// TwinCAT 3 PLC project SPS1
// ProgramVersion: 3.1.4023.0
// libraries:
//   Tc2_MC2, * (Beckhoff Automation GmbH)
//   Tc2_MC2_Drive, * (Beckhoff Automation GmbH)
//   Tc2_Standard, * (Beckhoff Automation GmbH)
//   Tc2_System, * (Beckhoff Automation GmbH)
//   Tc2_Utilities, * (Beckhoff Automation GmbH)
//   Tc3_Module, * (Beckhoff Automation GmbH)
//   Tc3_System, * (Beckhoff Automation GmbH)
// project tree:
//   DUTs/Standard/FunE/ u_FunEIF.TcDUT, u_FunEIF_In.TcDUT, u_FunEIF_InOut.TcDUT, u_FunEIF_Out.TcDUT, u_FunEIF_Stat.TcDUT
//   GVLs/Standard/ DB_FunE_IF.TcGVL, Globale_Konstanten.TcGVL
//   / PlcTask.TcTTO
//   POUs/ MAIN.TcPOU
//   POUs/Standardt/Hilfsfunktionen Zeit/ R_SYS_T.TcPOU, T_DIFF.TcPOU
//   POUs/Standardt/Zentral/ FB_Zentral.TcPOU, FB_Zentral_TaktimpulsGenerator.TcPOU
// real-time tasks:
//   TASK PlcTask: cycle T#10ms, priority 20, ADS port 350
// I/O:
//   DEVICE Gerät 1 (EtherCAT) (disabled), AmsNetId 192.168.27.57.2.1
//     Klemme 1 (EK1100) [EK1100 EtherCAT-Koppler (2A E-Bus)]
//       Klemme 2 (EL7201) [EL7201 1K. MDP742 Servo-Motor-Endstufe (50V, 4A)]

CONFIGURATION SPS1
    RESOURCE PLC ON TwinCAT3
        TASK PlcTask(INTERVAL := T#10ms, PRIORITY := 20);
        PROGRAM MAIN WITH PlcTask : MAIN;
    END_RESOURCE
END_CONFIGURATION

// ---- DUTs/Standard/FunE/u_FunEIF.TcDUT
TYPE u_FunEIF :
STRUCT
	I									:u_FunEIF_In; 
	O									:u_FunEIF_Out; 
	X									:u_FunEIF_InOut;
	Stat								:u_FunEIF_Stat;
END_STRUCT
END_TYPE

// ---- DUTs/Standard/FunE/u_FunEIF_In.TcDUT
TYPE u_FunEIF_In :
STRUCT
	x_Start									:BOOL := FALSE;															//Start Ablauf
	x_Init									:BOOL := FALSE; 														//Anwahl Initialisierung
	x_Freigabe							:BOOL := FALSE; 														//Freigabe Ablauf
	x_FreigabeHalt						:BOOL := FALSE; 														//Freigabe Unterbrechung
	x_FreigabeStoerung			:BOOL := FALSE; 														//Freigabe Stoerung
	x_FreigabeZeitEinlernen		:BOOL := FALSE; 														//Freigabe Ermittlung Regelzeit
	x_uFunEGST							:BOOL := FALSE; 														//unterlagerte Funktionselemente : alle in Grundstellungs
	x_uFunEinitAktiv					:BOOL := FALSE; 														//unterlagerte Funktionselemente: mind. 1 initialisierung aktiv 
	x_uFunEHalt							:BOOL := FALSE; 														//unterlagerte Funktionselemente: mind. 1 noch nicht fertig
	x_uFunEStoerung				:BOOL := FALSE; 														//unterlagerte Funktionselemente: mind. 1 hat Stoerung
	x_SimulationAktiv					:BOOL := FALSE; 														//Simulation aktiv
	i_Auftrag								:BOOL := FALSE; 														//Auftragsnummer
	t_Simulationszeit					:TIME := T#1S; 															//Verzögerungszeit für Simulation
	t_TimeOut							:TIME := T#1S; 															//TimeOut für Meldung wenn FunE länger braucht als eingelernt
	s_Name								:STRING := "Kein Funktionselement vergeben"; 		//Name des Funktionselements
	i_FunETyp							:INT := 0; 																	//Typ/Art des Funktionselements
	i_MasterFunE						:INT := 0; 																	//uebergeordnetes Funktionselement (bei 0 kein uebergeordnetes FunE)
END_STRUCT
END_TYPE

// ---- DUTs/Standard/FunE/u_FunEIF_InOut.TcDUT
TYPE u_FunEIF_InOut :
STRUCT
	x_Parameter					:ARRAY[0..255] OF BOOL; 
	di_Parameter					:ARRAY[0..31] OF DINT; 
	lr_Parameter					:ARRAY[0..31] OF LREAL; 
	s_Parameter					:ARRAY[0..1] OF STRING; 
END_STRUCT
END_TYPE

// ---- DUTs/Standard/FunE/u_FunEIF_Out.TcDUT
TYPE u_FunEIF_Out :
STRUCT
	x_bereit								:BOOL :=FALSE; 													//Funktionselement ist bereit
	x_arbeitet							:BOOL :=FALSE; 													//Funktionselement arbeitet
	x_fertig								:BOOL :=FALSE; 													//Funktionselement hat Zyklus beendet (steht bis zum nächsten Zyklus an)
	x_Fehler								:BOOL :=FALSE; 													//Funktionselement hat Fehler
	x_Grundstellung					:BOOL :=FALSE; 													//Funktionselement ist in Grundstellung
	x_initAktiv							:BOOL :=FALSE; 													//Funktionselement initialisierung aktiv 
	s_Aktionsname					:STRING :=""; 													//Name der aktuellen Aktion
	di_Status								:DINT := 0; 															//Statuscode (negativ=Fehler/positiv=erfolgreich)
	t_ZeitLetzerZyklus				:TIME := T#0MS; 												//Bearbeitungszeit letzter Ablauf
	di_Aktivierungen					:DINT := 0; 															//Anzahl der Aktivierungen 
	lt_Betriebsstundenzaehler 	:LTIME := LTIME#0MS; 										//Betriebsstundenzaehler
END_STRUCT
END_TYPE

// ---- DUTs/Standard/FunE/u_FunEIF_Stat.TcDUT
TYPE u_FunEIF_Stat :
STRUCT
	x_Halt												:BOOL :=FALSE; 								//FunE Halt
	x_Betrieb											:BOOL :=FALSE; 								//Betriebsfreigabe
	x_WSB												:BOOL :=FALSE;								//Weiterschaltbedingung
	x_Schrittwechsel								:BOOL :=FALSE; 								//Schrittwechsel aktiv
	i_SchrittFlanke									:INT :=0; 										//Schritt letzter SPS - Zyklus (benötigt zur Erkennung des Schrittwechsels)
	i_Schritt											:INT:= 0; 										//aktueller Schritt der Schrittkette
	i_SchrittAlt										:INT :=0; 										//letzter Schritt
	dt_StartZeit										:DT := DT#1972-03-29-00:00:00;	//Zeit, an dem das Funktionselement gestartet wurde	(Achtung!!!: In DT sind im gegensatz zu Siemens keine MS enthalten!!!)
	dt_LaufzeitFunE								:DT := DT#1972-03-29-00:00:00;  	//Zeit seit Start des Funktionselements (Achtung!!!: In DT sind im gegensatz zu Siemens keine MS enthalten!!!)
	t_mittlereZykluszeit							:TIME :=T#0MS; 								//eingelernte Zykluszeit
	o_Simulationszeit								:TON; 												//Timer für die Simulation des Funktionselements
END_STRUCT
END_TYPE

// ---- GVLs/Standard/DB_FunE_IF.TcGVL
{attribute 'qualified_only'}
VAR_GLOBAL
	Nr																	:ARRAY[0..Globale_Konstanten.Ci_Funktionselmente] OF u_FunEIF; 
	Anwahl_HMI_FunE_1									:INT :=0; 
	Anwahl_HMI_FunE_2									:INT :=0; 
	Anwahl_HMI_FunE_3									:INT :=0; 
	Anwahl_HMI_FunE_4									:INT :=0; 
END_VAR

// ---- GVLs/Standard/Globale_Konstanten.TcGVL
{attribute 'qualified_only'}
//Anwenderkonstanten
VAR_GLOBAL CONSTANT
	Ci_ZentralModuleAnzahl				:INT 		:=1; 					//Anzahl der autarken Zentralmodule
	Ci_Funktionselmente					:INT 		:=999; 				//Anzahl der Funktionselemente 
	Ci_Mod1										:INT			:=1; 					//EnumMR - Modul1
	Ci_Mod1RT1									:INT			:=1; 					//EnumMR - Modul1 RT1
END_VAR

// ---- POUs/MAIN.TcPOU
PROGRAM MAIN
VAR
	So_Taktgenerator				: FB_Zentral_TaktimpulsGenerator; 
	
	Sx_Takt			: BOOL; 
	Sx_Impuls		: BOOL; 
	Si_Counter		: INT; 
	
END_VAR


So_Taktgenerator(Ir_Frequenz := 1.0, Ox_Takt => Sx_Takt, Ox_Impuls => Sx_Impuls); 

IF(Sx_Impuls) THEN 
	Si_Counter := Si_Counter + 1;
END_IF

END_PROGRAM

// ---- POUs/Standardt/Zentral/FB_Zentral_TaktimpulsGenerator.TcPOU
FUNCTION_BLOCK FB_Zentral_TaktimpulsGenerator
VAR_INPUT
	Ir_Frequenz		: REAL; 
END_VAR
VAR_OUTPUT
	Ox_Takt								: BOOL; 
	Ox_Impuls							: BOOL; 
END_VAR

VAR
	St_TakttimerEinfach					: TON; 
	ReadRTC									: R_SYS_T; 
	TimeValid									: BOOL; 
	RTCTime									: DT; 
	RTCMillis									: DWORD; 
	Sdt_StartAktuellerTakt				: DT; 
	Sx_TaktFP								: BOOL; 
	Sx_Init										: BOOL; 
	St_DifferenzStartAktuell			:TIME; 	
	Sdw_StartAktuellerTaktMillis	:DWORD;  
END_VAR
	
VAR_TEMP

END_VAR

//Erfassung aktuelle Date and Time
ReadRTC(It_SynchTime := T#5S, Ox_TimeValid => TimeValid, Odt_RTCTime => RTCTime, Odw_Milliseconds => RTCMillis);  
	
//Ermittlung Dauer seit Taktstart
St_DifferenzStartAktuell := T_DIFF(Idt_Time1 := RTCTime, Idw_Time1Millis :=RTCMillis, Idt_Time2 := Sdt_StartAktuellerTakt, Idw_Time2Millis := Sdw_StartAktuellerTaktMillis); 


//Taktbildung (halbe Zeit an/ halbe Zeit aus)
Ox_Takt := St_DifferenzStartAktuell > DINT_TO_TIME(REAL_TO_DINT((1000/Ir_Frequenz)/2)); 
	
//Impuls Takt 
Ox_Impuls := Ox_Takt AND NOT Sx_TaktFP;
Sx_TaktFP := Ox_Takt; 
	
//Abspeichern Start aktueller Takt
IF (St_DifferenzStartAktuell > DINT_TO_TIME(REAL_TO_DINT((1000/Ir_Frequenz)))) OR NOT Sx_Init THEN 
	Sdt_StartAktuellerTakt := RTCTime; 
	Sdw_StartAktuellerTaktMillis := RTCMillis; 
END_IF
	
//Baustein als initialisiert setzen 
Sx_Init := TRUE;

END_FUNCTION_BLOCK

// ---- POUs/Standardt/Hilfsfunktionen Zeit/R_SYS_T.TcPOU
FUNCTION_BLOCK R_SYS_T
VAR_INPUT
	It_SynchTime						: TIME; 
END_VAR
VAR_OUTPUT
	Odt_RTCTime						: DT; 
	Odw_Milliseconds					: DWORD; 
	Ox_TimeValid						: BOOL; 
END_VAR
VAR
	So_SynchronizeTimer			: TON; 
	So_ReadSystemTime			: NT_GetTime; 
	Ss_SystemTime					: TIMESTRUCT; 
	Sx_Synch								: BOOL; 
	So_SynchTrigger					: F_TRIG; 
	So_RTC								: RTC_EX; 
	
	//Debug variables
	Si_SynchCounter					: DWORD; 
	
END_VAR

//Defines
{define DEBUG}

//Read System Time cyclic with period based on the Synch time 
So_SynchronizeTimer(IN := NOT So_SynchronizeTimer.Q, PT := It_SynchTime);
So_ReadSystemTime(START := So_SynchronizeTimer.Q,  TMOUT := DEFAULT_ADS_TIMEOUT, TIMESTR => Ss_SystemTime); 

//Create the synchronise bit
So_SynchTrigger(CLK := (So_ReadSystemTime.BUSY AND NOT So_ReadSystemTime.ERR)); 

//Count the Synchs in Debug Mode
{IF defined (DEBUG)}
	IF(So_SynchTrigger.Q) THEN 
		Si_SynchCounter := Si_SynchCounter + 1; 
	END_IF
{END_IF}

//RTC Synchronisieren und auslesen 
So_RTC(EN := So_SynchTrigger.Q, PDT := SYSTEMTIME_TO_DT(Ss_SystemTime), PMSEK := Ss_SystemTime.wMilliseconds, Q => Ox_TimeValid, CDT => Odt_RTCTime, CMSEK => Odw_Milliseconds);

END_FUNCTION_BLOCK

// ---- POUs/Standardt/Hilfsfunktionen Zeit/T_DIFF.TcPOU
FUNCTION T_DIFF : Time
VAR_INPUT
	Idt_Time1				:DT; 
	Idw_Time1Millis	:DWORD; 
	Idt_Time2				:DT; 
	Idw_Time2Millis	:DWORD; 
END_VAR
VAR
	Ss_Time1						:TIMESTRUCT;
	Ss_Time2						:TIMESTRUCT;
	Sw_HourDiff					:WORD; 
	Sw_MinuteDiff				:WORD; 
	Sw_SecondDiff				:WORD; 
	Sw_MillisecondsDiff		:DWORD;
	Sdw_TimeInMillis			:DWORD ; 
END_VAR

//Convert the time to TIMESTRUCT
Ss_Time1 := DT_TO_SYSTEMTIME(Idt_Time1); 
Ss_Time2 := DT_TO_SYSTEMTIME(Idt_Time2); 

//Subract
Sw_HourDiff := Ss_Time1.wHour - Ss_Time2.wHour; 
Sw_MinuteDiff := Ss_Time1.wMinute - Ss_Time2.wMinute; 
Sw_SecondDiff := Ss_Time1.wSecond - Ss_Time2.wSecond; 
Sw_MillisecondsDiff := Idw_Time1Millis - Idw_Time2Millis;

//Convert to millis
Sdw_TimeInMillis := Sdw_TimeInMillis + Sw_MillisecondsDiff; 
Sdw_TimeInMillis := Sdw_TimeInMillis + (Sw_SecondDiff*1000);
Sdw_TimeInMillis := Sdw_TimeInMillis + (Sw_MinuteDiff*1000*60); 
Sdw_TimeInMillis := Sdw_TimeInMillis + (Sw_HourDiff*1000*60*60); 

//Return 
T_DIFF := DWORD_TO_TIME(Sdw_TimeInMillis);

END_FUNCTION

// ---- POUs/Standardt/Zentral/FB_Zentral.TcPOU
FUNCTION_BLOCK FB_Zentral
VAR_INPUT
END_VAR
VAR_OUTPUT
END_VAR
VAR
END_VAR

END_FUNCTION_BLOCK
